Fanuc KAREL source: kd00041.KL

PROGRAM KD00041
%STACKSIZE=65535
%PRIORITY=65535
%NOLOCKGROUP
%ENVIRONMENT TPE
VAR
I : INTEGER
J : INTEGER
B : BOOLEAN
R : REAL
S : STRING[80]
-- UNRESOLVED DECLARATIONS (source type spelling not recovered)
-- D : TYPE_0x1100 (type_u16=0x1100)
BEGIN
I=1
END KD00041
